// TIA Portal V16 program export: 0 tag tables, 0 data types, 0 data blocks, 3 code blocks (in call order from the OBs), 0 instance data blocks

ORGANIZATION_BLOCK "Main"   // OB1, SCL, ProgramCycle
TITLE = "Main Program Sweep (Cycle)"
{ S7_Optimized_Access := 'TRUE' }
VERSION : 0.1
// stored: AutoNumber true, IsIECCheckEnabled false, SetENOAutomatically false
   VAR_INPUT
      Initial_Call : Bool;   // Initial call of this OB
      Remanence : Bool;   // =True, if remanent data are available
   END_VAR
BEGIN

   "MHJ-PLC-Lab-Function-S71500"(MinDiByte:=0,
                                 MaxDiByte:=1);
   "MHJ-PLC-Lab-Function-S71500-NextInputArea"(MinDiByte:=256,
                                               MaxDiByte:=259);


   "K1" := "S2";
   "K2" := "S3";
   "P5" := "S1";
   "P4" := "S4";
   "P3" := "S3";
   "P2" := NOT "S0";
   "P1" := "S3";
   "IstPos" := "SollPos";
END_ORGANIZATION_BLOCK

FUNCTION "MHJ-PLC-Lab-Function-S71500-NextInputArea" : Void   // FC2, SCL
{ S7_Optimized_Access := 'TRUE' }
VERSION : 0.1
// stored: AutoNumber true, IsIECCheckEnabled false, SetENOAutomatically false, UDAEnableTagReadback false
   VAR_INPUT
      MinDiByte : Int;
      MaxDiByte : Int;
   END_VAR
   VAR_TEMP
      Value : Byte;
      ForCounter : Int;
      MaxDiByteTemp : Int;
      MinDiByteTemp : Int;
   END_VAR
BEGIN


   #MaxDiByteTemp := -1;
   IF #MaxDiByte < 463 THEN
       #MaxDiByteTemp := #MaxDiByte;
   END_IF;

   #MinDiByteTemp := -1;
   IF #MaxDiByteTemp >= #MinDiByte & #MinDiByte >= 0 THEN
       #MinDiByteTemp := #MinDiByte;
   END_IF;

   IF #MaxDiByteTemp >= 0 & #MinDiByte >= 0 THEN
       FOR #ForCounter := #MinDiByteTemp TO #MaxDiByteTemp DO
           #Value := PEEK(area := 16#1,
                          dbNumber := 0,
                          byteOffset := #ForCounter);
           POKE(area := 16#81,
                dbNumber := 0,
                byteOffset := #ForCounter,
                value := #Value);
       END_FOR;

   END_IF;
END_FUNCTION

FUNCTION "MHJ-PLC-Lab-Function-S71500" : Void   // FC1, SCL
{ S7_Optimized_Access := 'TRUE' }
VERSION : 0.1
// stored: AutoNumber true, IsIECCheckEnabled false, SetENOAutomatically false, UDAEnableTagReadback false
   VAR_INPUT
      MinDiByte : Int;
      MaxDiByte : Int;
   END_VAR
   VAR_TEMP
      Value : Byte;
      ForCounter : Int;
      MaxDiByteTemp : Int;
      MinDiByteTemp : Int;
   END_VAR
   VAR CONSTANT
      Value_01_DW : DWord := 16#1223_5486;
      Value_02_DW : DWord := 16#A6C9_D1F5;
   END_VAR
BEGIN

   #Value:=PEEK(area := 16#82,
        dbNumber := 0,
        byteOffset := 511);
   #Value := #Value + 1;

   POKE(area := 16#82,
        dbNumber := 0,
        byteOffset := 511,
        value := #Value);

   POKE(area := 16#82,
        dbNumber := 0,
        byteOffset := 1016,
        value := #Value_01_DW);
   POKE(area := 16#82,
        dbNumber := 0,
        byteOffset := 1020,
        value := #Value_02_DW);

   #MaxDiByteTemp := 462;
   IF #MaxDiByte < 463 THEN
       #MaxDiByteTemp := #MaxDiByte;
   END_IF;

   #MinDiByteTemp := 0;
   IF #MaxDiByteTemp >= #MinDiByte & #MinDiByte >= 0 THEN
       #MinDiByteTemp := #MinDiByte;
   END_IF;

   FOR #ForCounter := #MinDiByteTemp TO #MaxDiByteTemp DO
       #Value := PEEK(area := 16#1,
                      dbNumber := 0,
                      byteOffset := #ForCounter);
       POKE(area := 16#81,
            dbNumber := 0,
            byteOffset := #ForCounter,
            value := #Value);
   END_FOR;

   #Value := PEEK(area := 16#1,
                  dbNumber := 0,
                  byteOffset := 512);
   POKE(area := 16#82,
        dbNumber := 0,
        byteOffset := 512,
        value := #Value);
END_FUNCTION
